// TwinCAT 3 PLC project Main_Control
// ProgramVersion: 3.1.4023.0
// libraries:
//   Tc2_Standard, * (Beckhoff Automation GmbH)
//   Tc2_System, * (Beckhoff Automation GmbH)
//   Tc3_Module, * (Beckhoff Automation GmbH)
// project tree:
//   / PlcTask.TcTTO
//   POUs/ MAIN.TcPOU
// real-time tasks:
//   TASK PlcTask: cycle T#10ms, priority 20, ADS port 350
// I/O:
//   DEVICE Device 1 (EtherCAT), AmsNetId 10.211.55.3.2.1
//     Term 1 (EK1200) [EK1200-7000 EtherCAT Power supply (1,5A E-Bus)]
//       Term 2 (EL1008) [EL1008 8Ch. Dig. Input 24V, 3ms]
//       Term 3 (EL1008) [EL1008 8Ch. Dig. Input 24V, 3ms]
//       Term 4 (EL1008) [EL1008 8Ch. Dig. Input 24V, 3ms]
//       Term 5 (EL3004) [EL3004 4Ch. Ana. Input +/-10V]
//       Term 6 (EL3004) [EL3004 4Ch. Ana. Input +/-10V]
//       Term 7 (EL9110) [EL9110 Power Supplier with LED (24V, Diagnostics)]
//       Term 8 (EL2008) [EL2008 8Ch. Dig. Output 24V, 0.5A]
//       Term 9 (EL2008) [EL2008 8Ch. Dig. Output 24V, 0.5A]
//       Term 10 (EL9110) [EL9110 Power Supplier with LED (24V, Diagnostics)]
//       Term 11 (EL2008) [EL2008 8Ch. Dig. Output 24V, 0.5A]
//       Term 12 (EL2008) [EL2008 8Ch. Dig. Output 24V, 0.5A]
//       Term 13 (EK1122) [EK1122 2 port EtherCAT junction]
//         Term 14 (EK1100) [EK1100 EtherCAT Coupler (2A E-Bus)]
//           Term 15 (EL1008) [EL1008 8Ch. Dig. Input 24V, 3ms]
//           Term 16 (EL1008) [EL1008 8Ch. Dig. Input 24V, 3ms]
//           Term 17 (EL9110) [EL9110 Power Supplier with LED (24V, Diagnostics)]
//           Term 18 (EL2008) [EL2008 8Ch. Dig. Output 24V, 0.5A]
//           Term 19 (EL2008) [EL2008 8Ch. Dig. Output 24V, 0.5A]

CONFIGURATION Main_Control
    RESOURCE PLC ON TwinCAT3
        TASK PlcTask(INTERVAL := T#10ms, PRIORITY := 20);
        PROGRAM MAIN WITH PlcTask : MAIN;
    END_RESOURCE
END_CONFIGURATION

// ---- POUs/MAIN.TcPOU
PROGRAM MAIN
VAR
END_VAR

END_PROGRAM
